{attribute 'linkalways'} 
{attribute 'no_explicit_call' := 'This FB is a CLASS and must be accessed using methods or properties'}
{attribute 'enable_dynamic_creation'}
FUNCTION_BLOCK _ETcVnConnectedComponentsAlgorithm EXTENDS EnumDatatypeBase
VAR
	localData : ETcVnConnectedComponentsAlgorithm;
	activeData : REFERENCE TO ETcVnConnectedComponentsAlgorithm;
	enumBaseDatatype : _DINT(localData);
END_VAR

METHOD PRIVATE AddLocalEnumeration
VAR_INPUT
	Enumeration : T_MAXSTRING;
	Value : ETcVnConnectedComponentsAlgorithm;
END_VAR
AddEnumeration(Enumeration, Value);
END_METHOD

PROPERTY PUBLIC Address : PVOID
GET
Address := ADR(activeData);
END_GET
END_PROPERTY

METHOD PUBLIC ClearReference
VAR_INPUT
END_VAR
activeData REF= localData;
SetBaseDatatypeReference();
END_METHOD

METHOD PUBLIC Clone : I_Datatype
VAR
    pClone : POINTER TO _ETcVnConnectedComponentsAlgorithm;
END_VAR
pClone := __NEW(_ETcVnConnectedComponentsAlgorithm(InitialValue := Value));
Clone := pClone^;
END_METHOD

METHOD FB_init : BOOL
VAR_INPUT
	bInitRetains : BOOL; // if TRUE, the retain variables are initialized (warm start / cold start)
	bInCopyCode : BOOL;  // if TRUE, the instance afterwards gets moved into the copy code (online change)
	InitialValue : ETcVnConnectedComponentsAlgorithm;
END_VAR
localData := InitialValue;
AddBaseDatatype(enumBaseDatatype);
ClearReference();

AddLocalEnumeration('TCVN_CCA_WU', ETcVnConnectedComponentsAlgorithm.TCVN_CCA_WU);
AddLocalEnumeration('TCVN_CCA_GRANA', ETcVnConnectedComponentsAlgorithm.TCVN_CCA_GRANA);
END_METHOD

PROPERTY PUBLIC Identifier : T_MAXSTRING
GET
Identifier := 'ETcVnConnectedComponentsAlgorithm';
END_GET
END_PROPERTY

METHOD IsEnumeratorValueEqual : BOOL
VAR_INPUT
	Enumerator : I_KeyValueForwardEnumerator;
END_VAR
VAR
	storedValue : ETcVnConnectedComponentsAlgorithm;
END_VAR
IF NOT Enumerator.TryGet(storedValue) THEN
	RETURN;
END_IF

IsEnumeratorValueEqual := storedValue = activeData;
END_METHOD

METHOD PUBLIC MakeReferenceTo
VAR_INPUT
	ReferenceTarget : REFERENCE TO ETcVnConnectedComponentsAlgorithm;
END_VAR
activeData REF= ReferenceTarget;
SetBaseDatatypeReference();
END_METHOD

METHOD PROTECTED SetBaseDatatypeReference
VAR_INPUT
END_VAR
enumBaseDatatype.MakeReferenceTo(activeData);
END_METHOD

PROPERTY PUBLIC Size : UDINT
GET
Size := SIZEOF(activeData);
END_GET
END_PROPERTY

METHOD TryMakeReferenceTo : BOOL
VAR_INPUT
	Target : I_Datatype;
END_VAR
VAR
	targetAsEnum : I_EnumDatatype;
	pTargetData : POINTER TO ETcVnConnectedComponentsAlgorithm;
END_VAR
IF NOT Target.TryResolveAsEnumDatatype(targetAsEnum) THEN
	RETURN;
END_IF

IF targetAsEnum.Identifier <> Identifier THEN
	RETURN;
END_IF

pTargetData := Target.Address;
activeData REF= pTargetData^;
SetBaseDatatypeReference();
TryMakeReferenceTo := TRUE;
END_METHOD

PROPERTY PUBLIC Value : ETcVnConnectedComponentsAlgorithm
GET
Value := activeData;
END_GET
SET
activeData := Value;
END_SET
END_PROPERTY

END_FUNCTION_BLOCK

(* stored: Version 1.1.0.1
   POU _ETcVnConnectedComponentsAlgorithm: Id {2fb3b48c-3725-489c-9093-fdcd0b387664}, SpecialFunc None
   Folder Constructor: Id {f361f57d-a9d2-4827-b253-0faa141f15c3}
   Folder Private: Id {2b36f8bd-25a9-4692-93e6-05fc540d3424}
   Folder Protected: Id {3df9f14e-1474-4f74-aa80-08a75c1ac695}
   Method AddLocalEnumeration: Id {ae6c35a8-438b-4f78-a650-ab254e4a09e7}
   Property Address: Id {974c10b0-d4c0-4363-abdb-0c11da01f3e8}
   Get Get: Id {e57b6ed3-4f1f-49c0-a739-e86a46871f70}
   Method ClearReference: Id {c7999bd6-b802-4066-931a-009f218ca3b2}
   Method Clone: Id {98fe0939-c6f0-435b-a31b-bf7a2be3d8a1}
   Method FB_init: Id {016d9ef3-dfa4-42cf-ac8a-de59bd98bc03}
   Property Identifier: Id {51529aaf-a897-46eb-b6cf-35d38645f438}
   Get Get: Id {bc83fb57-143d-4c6b-af44-e44e8479c7d1}
   Method IsEnumeratorValueEqual: Id {5d9fb4aa-790b-4584-87ce-2160475e6cca}
   Method MakeReferenceTo: Id {8e084b8f-0698-4280-87a3-ea4c3aa4263c}
   Method SetBaseDatatypeReference: Id {f817023d-5dc4-466b-9742-b557be31ab16}
   Property Size: Id {69a1056a-243b-401c-9856-e77d6059479e}
   Get Get: Id {f592bb55-00c2-443a-899f-910e8e2293bf}
   Method TryMakeReferenceTo: Id {997fed97-1f22-46a8-bdb1-b6f581165545}
   Property Value: Id {b2b0b62e-d493-4a26-b636-2a930a89f2f6}
   Get Get: Id {bf4eb79f-0931-45e0-b4eb-c659f39122ea}
   Set Set: Id {51c0da3b-34e3-4e7f-b3de-48d7db8aaf46} *)
